FUNCTION_BLOCK FB_Waermezaehler_MollineC3
VAR_INPUT
	Telegramm	: ARRAY[1..cMBUS_MaxTelegrams] OF ST_MBus_Data2;

END_VAR
VAR_IN_OUT
	Zustand		: ST_WZ_Zustand;
END_VAR
VAR
END_VAR
VAR // added by the converter: edge detectors and wires of the graphical bodies
    _w1, _w2 : ANY;
END_VAR

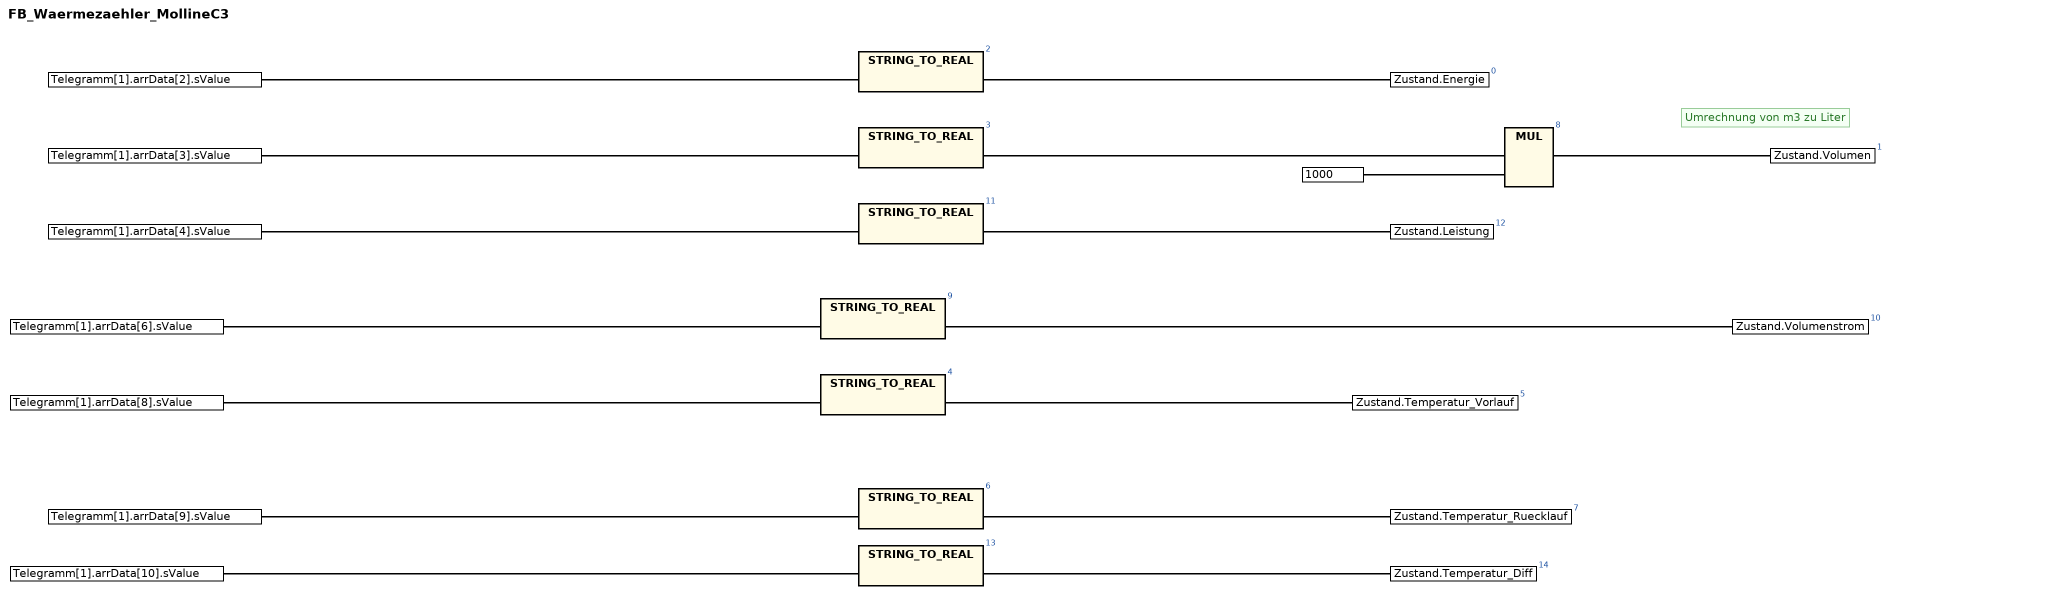
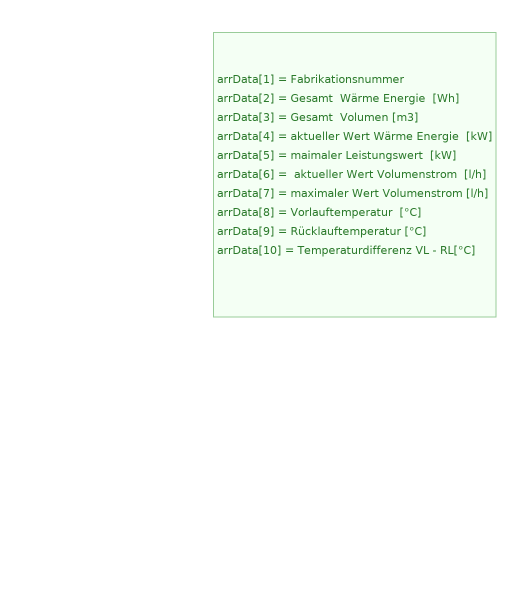
Zustand.Energie := _w1;
//
// arrData[1] = Fabrikationsnummer
// arrData[2] = Gesamt  Wärme Energie  [Wh]
// arrData[3] = Gesamt  Volumen [m3]
// arrData[4] = aktueller Wert Wärme Energie  [kW]
// arrData[5] = maimaler Leistungswert  [kW]
// arrData[6] =  aktueller Wert Volumenstrom  [l/h]
// arrData[7] = maximaler Wert Volumenstrom [l/h]
// arrData[8] = Vorlauftemperatur  [°C]
// arrData[9] = Rücklauftemperatur [°C]
// arrData[10] = Temperaturdifferenz VL - RL[°C]
//
//
//
// Umrechnung von m3 zu Liter
Zustand.Volumen := _w2;
_w1 := STRING_TO_REAL(Telegramm[1].arrData[2].sValue);
Zustand.Temperatur_Vorlauf := STRING_TO_REAL(Telegramm[1].arrData[8].sValue);
Zustand.Temperatur_Ruecklauf := STRING_TO_REAL(Telegramm[1].arrData[9].sValue);
_w2 := STRING_TO_REAL(Telegramm[1].arrData[3].sValue) * 1000;
Zustand.Volumenstrom := STRING_TO_REAL(Telegramm[1].arrData[6].sValue);
Zustand.Leistung := STRING_TO_REAL(Telegramm[1].arrData[4].sValue);
Zustand.Temperatur_Diff := STRING_TO_REAL(Telegramm[1].arrData[10].sValue);

END_FUNCTION_BLOCK

(* stored: Version 1.1.0.1, ProductVersion 3.1.4024.9
   POU FB_Waermezaehler_MollineC3: Id {76f84ade-572e-4275-8360-906944623512}, SpecialFunc None *)
